FUNCTION_BLOCK IN_CHOICE (* Drop-down WSTRING input *)
  (* Standard: 61499-1; Classification: GUI *)
  (* Version 0.2, 2002-05-03, JHC, Rockwell Automation, Made QI IV=true. *)
  (* Version 0.1, 2001-05-23, JHC, Rockwell Automation, XML version *)
  (* Version 0.0, 1998-12-15, JHC, Rockwell Automation, SRC version *)
  (* Compiler header: package fb.rt.hmi; *)
  (* Compiler Java IBM VisualAge 3.0 *)
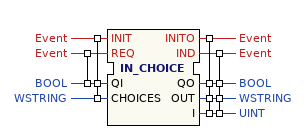
  EVENT_INPUT
    INIT WITH QI, CHOICES; (* Initialization *)
    REQ WITH QI; (* Request *)
  END_EVENT
  EVENT_OUTPUT
    INITO WITH QO, OUT, I; (* Initialization Confirm *)
    IND WITH QO, OUT, I; (* User changed choice or REQ serviced *)
  END_EVENT
  VAR_INPUT
    QI : BOOL := true; (* Event Qualifier *)
    CHOICES : WSTRING; (* Comma-separated list of choices *)
  END_VAR
  VAR_OUTPUT
    QO : BOOL; (* Event Qualifier *)
    OUT : WSTRING; (* Current Selection *)
    I : UINT; (* Index of Current Selection *)
  END_VAR
END_FUNCTION_BLOCK
